FUNCTION_BLOCK FB_DummyTool EXTENDS FB_MzTool
VAR_INPUT
END_VAR
VAR_OUTPUT
END_VAR

SUPER^();	//FB_MzTool aufrufen
aObjProcData[nNotifyId] := stProcessData;

ACTION A_Reset:
//Ist noch eine Aktion aktiv?
IF nStateA_ResetSpec = 0 THEN 
	nStateA_ResetSpec := 80;
END_IF

SUPER^.A_Reset();
END_ACTION

METHOD FB_init : BOOL
VAR_INPUT
	bInitRetains : BOOL; // if TRUE, the retain variables are initialized (warm start / cold start)
	bInCopyCode : BOOL;  // if TRUE, the instance afterwards gets moved into the copy code (online change)
END_VAR
eObjectType := E_ObjectType.OBJECTTYPE_DummyTool;
eObjectGroup := E_ObjectGroup.OBJECTGROUP_MzTool OR E_ObjectGroup.OBJECTGROUP_Device;
END_METHOD

END_FUNCTION_BLOCK

(* stored: Version 1.1.0.1, ProductVersion 3.1.4024.11
   POU FB_DummyTool: Id {e289cb84-c429-4034-9a3e-6c4d0ba27c7b}, SpecialFunc None
   Action A_Reset: Id {0e107c39-5304-4a4b-983f-052c8cd0d723}
   Method FB_init: Id {3f39baf6-5156-4236-9c57-0b118ee8823a} *)
